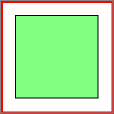
VISUALIZATION VisuMover  // 114x114
VAR_INPUT
	i : INT;
	
END_VAR
    RoundedRectangle (0,0 114x114), "%d", text variable: i
        p3560616238: MAIN.XPlanar1.Movers[i]._Mover.stMoverRef.MCTOPLC.ACT.ActPos.x
        p2738717112: GVL.iVisuYoffset-MAIN.XPlanar1.Movers[i]._Mover.stMoverRef.MCTOPLC.ACT.ActPos.y
        p2858320360: -MAIN.XPlanar1.Movers[i]._Mover.stMoverRef.MCTOPLC.ACT.ActPos.c
    RoundedRectangle (15,15 83x83), colour toggle: GVL.MoverProcessData[i].Status>=99, invisible if: MAIN.MoverProcessData[i].Status=0
        p3560616238: MAIN.XPlanar1.Movers[i]._Mover.stMoverRef.MCTOPLC.ACT.ActPos.x
        p2738717112: GVL.iVisuYoffset-MAIN.XPlanar1.Movers[i]._Mover.stMoverRef.MCTOPLC.ACT.ActPos.y
        p2858320360: -MAIN.XPlanar1.Movers[i]._Mover.stMoverRef.MCTOPLC.ACT.ActPos.c
        OnMouseClick: execute { GVL.MoverProcessData[i].Status:=99; }
END_VISUALIZATION

(* stored: Version 1.1.0.1, ProductVersion 3.1.4024.12
   Visu VisuMover: Id {0d3aa3ac-ecd2-442b-ae0e-3d6009cc9db4} *)
